(* CODESYS project Damper.library
   TcLibraryId: TE140x Module Vendor|Damper|0.0.0.2
   Company: TE140x Module Vendor
   DefaultNamespace: Damper
   Version: 0.0.0.2
   Placeholder: Damper
   Title: Damper

Project tree, tasks and I/O mapping:
  Version/
    global variables Global_Version
  POUs/
    function block FB_Damper [ST]: FB_exit, FB_init, nHResult, eInitExceptionHandling, eUpdateExceptionHandling, nExceptionCnt, stActiveException, bInitialized, bExecute
  DUTs/
    data type ST_FB_Damper_FB_Main
    data type ST_FB_Damper_FB_exit
    data type ST_FB_Damper_FB_init
    data type ST_GetSet_HRESULT
    data type E_FpExcptCtrlSetEx
    data type ST_GetSet_E_FpExcptCtrlSetEx
    data type ST_GetSet_ULINT
    data type ST_ExceptionInfo
    data type ST_GetSet_ST_ExceptionInfo
    data type ST_GetSet_BOOL
    data type ST_B_Damper_T
    data type ST_ExtU_Damper_T
    data type ST_ExtY_Damper_T
    data type ST_P_Damper_T
    data type ST_XDis_Damper_T
    data type ST_X_Damper_T
*)

// DUTs/ST_FB_Damper_FB_Main

	{attribute 'TcIecLibraryType'}
{attribute 'hide'}
TYPE ST_FB_Damper_FB_Main : 
	STRUCT
		 {attribute 'GUID' := '18071995-0000-0000-0000-000000000018'}
		pInst : PVOID;
		result : BOOL;
		 {attribute 'hide'}
		_reserved1 : UINT_24_56;
	END_STRUCT
END_TYPE

// DUTs/ST_FB_Damper_FB_exit

	{attribute 'TcIecLibraryType'}
{attribute 'hide'}
TYPE ST_FB_Damper_FB_exit : 
	STRUCT
		 {attribute 'GUID' := '18071995-0000-0000-0000-000000000018'}
		pInst : PVOID;
		bInCopyCode : BOOL;
		result : BOOL;
		 {attribute 'hide'}
		_reserved1 : UINT_16_48;
	END_STRUCT
END_TYPE

// DUTs/ST_FB_Damper_FB_init

	{attribute 'TcIecLibraryType'}
{attribute 'hide'}
TYPE ST_FB_Damper_FB_init : 
	STRUCT
		 {attribute 'GUID' := '18071995-0000-0000-0000-000000000018'}
		pInst : PVOID;
		bInitRetains : BOOL;
		bInCopyCode : BOOL;
		result : BOOL;
		 {attribute 'hide'}
		_reserved1 : UINT_8_40;
	END_STRUCT
END_TYPE

// DUTs/ST_GetSet_HRESULT

	{attribute 'TcIecLibraryType'}
{attribute 'hide'}
TYPE ST_GetSet_HRESULT : 
	STRUCT
		 {attribute 'GUID' := '18071995-0000-0000-0000-000000000018'}
		pInst : PVOID;
		 {attribute 'GUID' := '18071995-0000-0000-0000-000000000019'}
		nParam : HRESULT;
		 {attribute 'hide'}
		_reserved1 : UINT_0_32;
	END_STRUCT
END_TYPE

// DUTs/E_FpExcptCtrlSetEx

(* Generated from type 'TcMgSdk.FpExcptCtrlSetEx' *)
	{attribute 'TcIecLibraryType'}
TYPE E_FpExcptCtrlSetEx : (
	CallerExceptions:=1, 	(* Use the floating point exception settings provided by the caller *)
	ThrowExceptions:=3, 	(* Enable floating point exceptions on invalid operations and divisions by zero *)
	SuppressExceptions:=13, 	(* Disable floating point exceptions. *)
	LogExceptions:=19, 	(* Log exception information. *)
	LogAndHold:=51, 	(* Log exception information and puase execution of the cyclic code after completion of the actual cycle *)
	LogAndCatch:=83, 	(* Log exception information and immediately terminate execution of the cyclic code. Reinitialization is required to restart. *)
	LogAndDump:=147, 	(* Log exception information, create a dump file with detailed exception information and try to continue execution of the cyclic code *)
	LogHoldAndDump:=179, 	(* Log exception information, create a dump file with detailed exception information and puase execution of the cyclic code after completion of the actual cycle *)
	LogCatchAndDump:=211	(* Log exception information, create a dump file with detailed exception information and immediately terminate execution of the cyclic code. Reinitialization is required to restart. *)
) USINT;
END_TYPE

// DUTs/ST_GetSet_E_FpExcptCtrlSetEx

	{attribute 'TcIecLibraryType'}
{attribute 'hide'}
TYPE ST_GetSet_E_FpExcptCtrlSetEx : 
	STRUCT
		 {attribute 'GUID' := '18071995-0000-0000-0000-000000000018'}
		pInst : PVOID;
		eParam : E_FpExcptCtrlSetEx;
		 {attribute 'hide'}
		_reserved1 : UINT_24_56;
	END_STRUCT
END_TYPE

// DUTs/ST_GetSet_ULINT

	{attribute 'TcIecLibraryType'}
{attribute 'hide'}
TYPE ST_GetSet_ULINT : 
	STRUCT
		 {attribute 'GUID' := '18071995-0000-0000-0000-000000000018'}
		pInst : PVOID;
		nParam : ULINT;
	END_STRUCT
END_TYPE

// DUTs/ST_ExceptionInfo

(* Generated from type 'TcMgSdk.ExceptionInfo' *)
	{attribute 'TcIecLibraryType'}
TYPE ST_ExceptionInfo : 
	STRUCT
		(* Generated from item 'ExceptionCode' *)
		nExceptionCode : DINT;
		(* Generated from item 'TmxName' *)
		 {attribute 'GUID' := '18071995-0000-0000-0000-00010000007F'}
		sTmxName : STRING(127);
		(* Generated from item 'TmxVersion' *)
		nTmxVersion : ARRAY [0..3] OF UDINT;
		(* Generated from item 'InstructionAddr' *)
		nInstructionAddr : UDINT;
		(* Generated from item 'ReturnAddr' *)
		nReturnAddr : ARRAY [0..3] OF UDINT;
		(* Generated from item 'DumpCreated' *)
		bDumpCreated : BOOL;
		 {attribute 'hide'}
		_reserved1 : ARRAY [1..3] OF USINT;
	END_STRUCT
END_TYPE

// DUTs/ST_GetSet_ST_ExceptionInfo

	{attribute 'TcIecLibraryType'}
{attribute 'hide'}
TYPE ST_GetSet_ST_ExceptionInfo : 
	STRUCT
		 {attribute 'GUID' := '18071995-0000-0000-0000-000000000018'}
		pInst : PVOID;
		stParam : ST_ExceptionInfo;
		 {attribute 'hide'}
		_reserved1 : UINT_0_32;
	END_STRUCT
END_TYPE

// DUTs/ST_GetSet_BOOL

	{attribute 'TcIecLibraryType'}
{attribute 'hide'}
TYPE ST_GetSet_BOOL : 
	STRUCT
		 {attribute 'GUID' := '18071995-0000-0000-0000-000000000018'}
		pInst : PVOID;
		bParam : BOOL;
		 {attribute 'hide'}
		_reserved1 : UINT_24_56;
	END_STRUCT
END_TYPE

// DUTs/ST_B_Damper_T

(* Generated from type 'B_Damper_T' *)
	{attribute 'TcIecLibraryType'}
TYPE ST_B_Damper_T : 
	STRUCT
		(* Generated from item 'FilterCoefficient' *)
		fFilterCoefficient : LREAL;
		(* Generated from item 'SumI4' *)
		fSumI4 : LREAL;
		(* Generated from item 'Integrator' *)
		fIntegrator : LREAL;
		(* Generated from item 'IntegralGain' *)
		fIntegralGain : LREAL;
		(* Generated from item 'Saturation' *)
		fSaturation : LREAL;
		(* Generated from item 'Gain1' *)
		fGain1 : LREAL;
		(* Generated from item 'Kb' *)
		fKb : LREAL;
	END_STRUCT
END_TYPE

// DUTs/ST_ExtU_Damper_T

(* Generated from type 'ExtU_Damper_T' *)
	{attribute 'TcIecLibraryType'}
TYPE ST_ExtU_Damper_T : 
	STRUCT
		(* Generated from item 'struct_acc' *)
		fstruct_acc : LREAL;
	END_STRUCT
END_TYPE

// DUTs/ST_ExtY_Damper_T

(* Generated from type 'ExtY_Damper_T' *)
	{attribute 'TcIecLibraryType'}
TYPE ST_ExtY_Damper_T : 
	STRUCT
		(* Generated from item 'cart_acc' *)
		fcart_acc : LREAL;
	END_STRUCT
END_TYPE

// DUTs/ST_P_Damper_T

(* Generated from type 'P_Damper_T' *)
	{attribute 'TcIecLibraryType'}
TYPE ST_P_Damper_T : 
	STRUCT
		(* Generated from item 'cart_mass' *)
		fcart_mass : LREAL;
		(* Generated from item 'structure_mass' *)
		fstructure_mass : LREAL;
		(* Generated from item 'PIDController_D' *)
		fPIDController_D : LREAL;
		(* Generated from item 'PIDController_I' *)
		fPIDController_I : LREAL;
		(* Generated from item 'PIDController_InitialConditionF' *)
		fPIDController_InitialConditionF : LREAL;
		(* Generated from item 'PIDController_InitialConditio_e' *)
		fPIDController_InitialConditio_e : LREAL;
		(* Generated from item 'PIDController_Kb' *)
		fPIDController_Kb : LREAL;
		(* Generated from item 'PIDController_LowerSaturationLi' *)
		fPIDController_LowerSaturationLi : LREAL;
		(* Generated from item 'PIDController_N' *)
		fPIDController_N : LREAL;
		(* Generated from item 'PIDController_P' *)
		fPIDController_P : LREAL;
		(* Generated from item 'PIDController_UpperSaturationLi' *)
		fPIDController_UpperSaturationLi : LREAL;
	END_STRUCT
END_TYPE

// DUTs/ST_XDis_Damper_T

(* Generated from type 'XDis_Damper_T' *)
	{attribute 'TcIecLibraryType'}
TYPE ST_XDis_Damper_T : 
	STRUCT
		(* Generated from item 'Integrator_CSTATE' *)
		bIntegrator_CSTATE : BOOL;
		(* Generated from item 'Filter_CSTATE' *)
		bFilter_CSTATE : BOOL;
	END_STRUCT
END_TYPE

// DUTs/ST_X_Damper_T

(* Generated from type 'X_Damper_T' *)
	{attribute 'TcIecLibraryType'}
TYPE ST_X_Damper_T : 
	STRUCT
		(* Generated from item 'Integrator_CSTATE' *)
		fIntegrator_CSTATE : LREAL;
		(* Generated from item 'Filter_CSTATE' *)
		fFilter_CSTATE : LREAL;
	END_STRUCT
END_TYPE

// Version/Global_Version
{attribute 'TcGenerated'}
// This function has been automatically generated from the project information.
VAR_GLOBAL CONSTANT
	{attribute 'const_non_replaced'}
	{attribute 'linkalways'}
	stLibVersion_Damper : ST_LibVersion := (iMajor := 0, iMinor := 0, iBuild := 0, iRevision := 2, sVersion := '0.0.0.2');
	{attribute 'const_non_replaced'}
	{attribute 'linkalways'}
	sLibraryId_Damper : String := 'TE140x Module Vendor|Damper|0.0.0.2';
END_VAR

// POUs/FB_Damper

	{attribute 'c++_compatible'}
	{attribute 'external_name' := 'FB_Damper_GUID_3082C189_7AEE_E832_FAB6_F7C054266251'}
	{attribute 'TcIecLibraryType'}
	{attribute 'reflection'}
	FUNCTION_BLOCK FB_Damper
	VAR
		{attribute 'hide'}
		{attribute 'no_copy'}
		 {attribute 'GUID' := '18071995-0000-0000-0000-000000000018'}
		m_pData : PVOID;
		{attribute 'TcInitSymbol'}
		 {attribute 'GUID' := '8007AE3B-86BB-40F2-B385-EF87FCC239A4'}
		eTraceLevelMax : TcTraceLevel := TcTraceLevel.tlInfo;
		 {attribute 'hide'}
		_reserved1 : UDINT;
		{attribute 'hide'}
		{attribute 'instance-path'}
		{attribute 'noinit'}
		 {attribute 'GUID' := '18071995-0000-0000-0000-0001000000FF'}
		sInstancePath : STRING(255);
		{attribute 'hide'}
		{attribute 'noinit'}
		 {attribute 'GUID' := '18071995-0000-0000-0000-000000000019'}
		m_HResultLog : HRESULT;
		{attribute 'hide'}
		{attribute 'noinit'}
		 {attribute 'GUID' := '18071995-0000-0000-0000-000000000019'}
		m_HResult : HRESULT;
		 {attribute 'hide'}
		_reserved2 : ARRAY [1..184] OF USINT;
		{attribute 'hide'}
		{attribute 'no_copy'}
		m_ExtModeData : ULINT;
	END_VAR
	VAR_INPUT
		(* Generated from item 'struct_acc' *)
		fstruct_acc : LREAL;
	END_VAR
	VAR_OUTPUT
		(* Generated from item 'cart_acc' *)
		fcart_acc : LREAL;
	END_VAR
	VAR
		(* Generated from item 'PDamper_M' *)
		 {attribute 'GUID' := '18071995-0000-0000-0000-000000000018'}
		pPDamper_M : PVOID;
	END_VAR


	METHOD FB_exit : BOOL
	VAR_INPUT
		bInCopyCode : BOOL;
	END_VAR
END_METHOD


	METHOD FB_init : BOOL
	VAR_INPUT
		bInitRetains : BOOL;
		bInCopyCode : BOOL;
	END_VAR
END_METHOD


{attribute 'monitoring' := 'call'}
	PROPERTY nHResult : HRESULT
GET
END_GET
END_PROPERTY


{attribute 'monitoring' := 'call'}
	PROPERTY eInitExceptionHandling : E_FpExcptCtrlSetEx
GET
END_GET
SET
END_SET
END_PROPERTY


{attribute 'monitoring' := 'call'}
	PROPERTY eUpdateExceptionHandling : E_FpExcptCtrlSetEx
GET
END_GET
SET
END_SET
END_PROPERTY


{attribute 'monitoring' := 'call'}
	PROPERTY nExceptionCnt : ULINT
GET
END_GET
END_PROPERTY


{attribute 'monitoring' := 'variable'}
	PROPERTY stActiveException : ST_ExceptionInfo
GET
END_GET
END_PROPERTY


{attribute 'monitoring' := 'call'}
	PROPERTY bInitialized : BOOL
GET
END_GET
END_PROPERTY


{attribute 'monitoring' := 'call'}
	PROPERTY bExecute : BOOL
GET
END_GET
SET
END_SET
END_PROPERTY

END_FUNCTION_BLOCK
